// TIA Portal V20 export
DATA_BLOCK "GDB_MachineCmd"   // DB1
TITLE = Machine command/status DB
{ S7_Optimized_Access := 'TRUE' }
// Wang Shuo / Huashili-style command + status struct for ABCDE auto cycle. HMI binds buttons here.
// stored: MemoryReserve 100
   VAR
      bo_InitPath : Bool;   // HMI: rising edge → initialize ABCDE 5-point path data
      bo_Start : Bool;   // HMI: rising edge → start auto cycle (i16_AutoStep := 10)
      bo_Stop : Bool;   // HMI: rising edge → stop auto cycle (i16_AutoStep := 0)
      bo_Mode : Bool := TRUE;   // HMI: AUTO mode selector (TRUE = auto cycle enabled, FALSE = ignored)
      bo_ESTOP_LOCK : Bool := TRUE;   // Safety: E-Stop chain healthy (TRUE = OK, FALSE = E-Stop active)
      bo_PathInitialed : Bool;   // Status: ABCDE path has been initialized (set after bo_InitPath rising edge)
      bo_Alarm : Bool;   // Status: any system alarm (placeholder, always FALSE in minimal demo)
      i16_AutoStep : Int;   // Main state machine step. 6-state per source spec 杨子楠5月17日周计划.md §3.3: 0=idle, 10=going-to-A, 20=going-to-B, 30=going-to-C, 40=going-to-D, 50=going-to-E. Cycle wraps 50→10 (source spec §3.5). Wang Shuo / Huashili 4-REGION pattern.
   END_VAR
BEGIN
END_DATA_BLOCK
